
FUNCTION CB_sub_time : TIME


TITLE = ' Substracting two duration '
VERSION : '1.0'
AUTHOR  : CB
NAME    : sub_time
FAMILY  : TNI

VAR_INPUT
    IN0 : TIME;
    IN1 : TIME;
END_VAR

BEGIN
    CB_sub_time := IN0 - IN1;
END_FUNCTION
